//==============================================================
// 12) Brake release control
//==============================================================
// EN: A movement request keeps the magnetic brake released.
//     After movement stops, the brake remains released for a hold time.
conveyorLevelerMoveRequest :=
    systemRunEnable AND
    safetyCircuitOk AND
    conveyorLevelerDriveOk AND
    NOT conveyorLevelerFault AND
    (ABS(conveyorLevelerSignedSpeedRefMmps) >= machineConfig.conveyorLevelerRunMinSpeedMmps);


IF conveyorLevelerMoveRequest THEN

    conveyorLevelerBrakeReleaseRequest := TRUE;

    tonConveyorLevelerBrakeHoldDelay(IN := FALSE);

ELSE

    IF conveyorLevelerBrakeRelease THEN

        tonConveyorLevelerBrakeHoldDelay(
            IN := TRUE,
            PT := machineConfig.conveyorLevelerBrakeHoldTime
        );

        conveyorLevelerBrakeReleaseRequest :=
            NOT tonConveyorLevelerBrakeHoldDelay.Q;

    ELSE

        tonConveyorLevelerBrakeHoldDelay(IN := FALSE);
        conveyorLevelerBrakeReleaseRequest := FALSE;

    END_IF

END_IF;


conveyorLevelerBrakeRelease :=
    systemRunEnable AND
    safetyCircuitOk AND
    conveyorLevelerDriveOk AND
    NOT conveyorLevelerFault AND
    conveyorLevelerBrakeReleaseRequest;


//==============================================================
// 13) Brake release delay before motor movement
//==============================================================
// EN: The motor can run only after brake release delay.
tonConveyorLevelerBrakeReleaseDelay(
    IN := conveyorLevelerMoveRequest AND conveyorLevelerBrakeRelease,
    PT := machineConfig.conveyorLevelerBrakeReleaseDelay
);


//==============================================================
// 14) Conveyor leveler direction and speed outputs
//==============================================================
// EN: Convert signed internal speed command into direction outputs
//     and positive speed reference.
IF conveyorLevelerMoveRequest AND
   conveyorLevelerBrakeRelease AND
   tonConveyorLevelerBrakeReleaseDelay.Q THEN

    conveyorLevelerSpeedRefMmps :=
        ABS(conveyorLevelerSignedSpeedRefMmps);

    conveyorLevelerRunUp :=
        conveyorLevelerSignedSpeedRefMmps > 0.0;

    conveyorLevelerRunDown :=
        conveyorLevelerSignedSpeedRefMmps < 0.0;

ELSE

    conveyorLevelerSpeedRefMmps := 0.0;

    conveyorLevelerRunUp := FALSE;
    conveyorLevelerRunDown := FALSE;

END_IF;
END_METHOD

//==============================================================
// SIMPLE STACKER — SPEED REFERENCE GENERATOR
// EN: Generates synchronized and sheet-stack separation speed references [m/min].
//==============================================================
METHOD _ConveyorSpeedControl
VAR
    rPackageComplete                  : BOOL;
    packageGapReady                   : BOOL;
    validCycleTimeS                   : REAL;

    sheetConveyorsSpeedUpReferenceMPM : REAL;

    sheetConveyor1BaseSpeedMPM        : REAL;
    sheetConveyor2BaseSpeedMPM        : REAL;
    sheetConveyor3BaseSpeedMPM        : REAL;
END_VAR


//==============================================================
// 1) Default event pulses
//==============================================================
sheetStackSeparationStarted         := FALSE;
sheetStackSeparationFinished        := FALSE;

sheetConveyor2SeparationStarted     := FALSE;
sheetConveyor2SeparationFinished    := FALSE;

sheetConveyor3SeparationStarted     := FALSE;
sheetConveyor3SeparationFinished    := FALSE;


//==============================================================
// 2) Edge detection
//==============================================================
rPackageComplete := packageCompleteCmd AND NOT packageCompleteCmdOld;
packageCompleteCmdOld := packageCompleteCmd;


//==============================================================
// 3) Enable and scan time
//==============================================================
speedControlEnabled :=
    sheetConveyor1Run AND
    sheetConveyor2Run AND
    sheetConveyor3Run AND
    safetyCircuitOk;

rampReset := NOT speedControlEnabled;


// EN: Read PLC scan time using OSCAT CYCLE_TIME.
instCycleTime(
    RST := resetCmd
);


// EN: Convert last cycle time from TIME/ms to seconds.
scanTimeMs := TIME_TO_REAL(instCycleTime.ct_last);

validCycleTimeS :=
    LIMIT(
        0.001,
        scanTimeMs / 1000.0,
        20.0
    );

scanTimeS := validCycleTimeS;



//==============================================================
// 4) Calculate normal stacker speed
//==============================================================
IF speedControlEnabled THEN

    normalStackerSpeedMPM :=
        LIMIT(
            machineConfig.minimumSpeedMPM,
            MAX(0.0, lineSpeedMPM) *
                MAX(0.0, machineConfig.stackerSpeedRatio),
            machineConfig.maximumSpeedMPM
        );

ELSE

    normalStackerSpeedMPM := 0.0;

END_IF;


//==============================================================
// 6) Calculate normal speed for each conveyor
//==============================================================
sheetConveyor1NormalSpeedMPM :=
    normalStackerSpeedMPM *
    MAX(0.0, machineConfig.sheetConveyor1SpeedTrim);

sheetConveyor2NormalSpeedMPM :=
    normalStackerSpeedMPM *
    MAX(0.0, machineConfig.sheetConveyor2SpeedTrim);

sheetConveyor3NormalSpeedMPM :=
    normalStackerSpeedMPM *
    MAX(0.0, machineConfig.sheetConveyor3SpeedTrim);


//==============================================================
// 6.1) Sheet conveyors speed-up reference
//==============================================================
// EN: Speed-up is added directly to conveyors 1/2/3 references.
//     It can work even when line speed is zero, as long as the
//     conveyor group is enabled.
IF speedControlEnabled AND sheetConveyorsSpeedUpCmd THEN

    sheetConveyorsSpeedUpReferenceMPM :=
        MAX(0.0, machineConfig.sheetConveyorsSpeedUpMPM);

ELSE

    sheetConveyorsSpeedUpReferenceMPM := 0.0;

END_IF;


//==============================================================
// 6.2) Base speed references including speed-up
//==============================================================
// EN: Base speed is the synchronized conveyor speed plus operator speed-up.
//     Separation tracking must use this base speed as reference.
sheetConveyor1BaseSpeedMPM :=
    sheetConveyor1NormalSpeedMPM + sheetConveyorsSpeedUpReferenceMPM;

sheetConveyor2BaseSpeedMPM :=
    sheetConveyor2NormalSpeedMPM + sheetConveyorsSpeedUpReferenceMPM;

sheetConveyor3BaseSpeedMPM :=
    sheetConveyor3NormalSpeedMPM + sheetConveyorsSpeedUpReferenceMPM;


//==============================================================
// 7) Calculate separation high speed
//==============================================================
// EN: Gap speed also receives the same speed-up reference.
//     This preserves the real gap differential while allowing operator boost.
sheetConveyor2GapSpeedMPM :=
    (sheetConveyor2NormalSpeedMPM * MAX(0.0, machineConfig.packageGapSpeedRatio)) +
    machineConfig.packageGapSpeedOffsetMPM +
    sheetConveyorsSpeedUpReferenceMPM;

sheetConveyor3GapSpeedMPM :=
    (sheetConveyor3NormalSpeedMPM * MAX(0.0, machineConfig.packageGapSpeedRatio)) +
    machineConfig.packageGapSpeedOffsetMPM +
    sheetConveyorsSpeedUpReferenceMPM;


//==============================================================
// 8) Calculate separation tracking target distances
//==============================================================
// EN: Separation tracking target is based on each conveyor length.
sheetConveyor2TargetDistanceM :=
    MAX(0.0, machineConfig.sheetConveyor2LengthM);

sheetConveyor3TargetDistanceM :=
    MAX(0.0, machineConfig.sheetConveyor3LengthM);


//==============================================================
// 9) Check separation ready conditions
//==============================================================
// EN: Compare gap speed against base speed, not normal speed.
//     Otherwise operator speed-up would be incorrectly counted as gap opening.
packageGapReady :=
    speedControlEnabled AND
    (sheetConveyor2TargetDistanceM > 0.0) AND
    (sheetConveyor3TargetDistanceM > 0.0) AND
    ((sheetConveyor2GapSpeedMPM - sheetConveyor2BaseSpeedMPM) >= machineConfig.minimumOpeningSpeedMPM) AND
    ((sheetConveyor3GapSpeedMPM - sheetConveyor3BaseSpeedMPM) >= machineConfig.minimumOpeningSpeedMPM);

sheetStackSeparationReady := packageGapReady;


//==============================================================
// 10) Sheet stack separation state machine
//==============================================================
IF NOT speedControlEnabled THEN

    sheetStackSeparationState      := 'DISABLED';
    sheetStackSeparationStateCode  := -1;

    packageSeparationState         := 0;

    sheetStackSeparationActive     := FALSE;
    sheetStackBrakeActive          := FALSE;
    brakeValve                     := FALSE;

    sheetConveyor2SeparationActive := FALSE;
    sheetConveyor3SeparationActive := FALSE;

    sheetConveyor2HighSpeedActive  := FALSE;
    sheetConveyor3HighSpeedActive  := FALSE;

    sheetConveyor2OpeningDistanceM := 0.0;
    sheetConveyor3OpeningDistanceM := 0.0;

    sheetConveyor1TargetSpeedMPM   := 0.0;
    sheetConveyor2TargetSpeedMPM   := 0.0;
    sheetConveyor3TargetSpeedMPM   := 0.0;


ELSE

    CASE packageSeparationState OF

        0: // NORMAL
            sheetStackSeparationState     := 'NORMAL';
            sheetStackSeparationStateCode := 0;

            sheetStackSeparationActive    := FALSE;
            sheetStackBrakeActive         := FALSE;
            brakeValve                    := FALSE;

            sheetConveyor2SeparationActive := FALSE;
            sheetConveyor3SeparationActive := FALSE;

            sheetConveyor2HighSpeedActive  := FALSE;
            sheetConveyor3HighSpeedActive  := FALSE;

            sheetConveyor2OpeningDistanceM := 0.0;
            sheetConveyor3OpeningDistanceM := 0.0;

            sheetConveyor1TargetSpeedMPM  := sheetConveyor1BaseSpeedMPM;
            sheetConveyor2TargetSpeedMPM  := sheetConveyor2BaseSpeedMPM;
            sheetConveyor3TargetSpeedMPM  := sheetConveyor3BaseSpeedMPM;

            IF rPackageComplete AND packageGapReady THEN
                packageSeparationState := 10;
            END_IF


        10: // START_SHEET_STACK_SEPARATION
            sheetStackSeparationState     := 'START_SEPARATION';
            sheetStackSeparationStateCode := 10;

            sheetStackSeparationActive    := TRUE;
            sheetStackSeparationStarted   := TRUE;

            sheetStackBrakeActive         := TRUE;
            brakeValve                    := TRUE;

            // EN: Conveyor 2 tracking starts immediately.
            sheetConveyor2SeparationStarted := TRUE;

            sheetConveyor2SeparationActive  := TRUE;
            sheetConveyor3SeparationActive  := FALSE;

            // EN: Conveyor 2 and 3 accelerate together from the beginning.
            sheetConveyor2HighSpeedActive   := TRUE;
            sheetConveyor3HighSpeedActive   := TRUE;

            sheetConveyor2OpeningDistanceM  := 0.0;
            sheetConveyor3OpeningDistanceM  := 0.0;

            sheetConveyor1TargetSpeedMPM    := sheetConveyor1BaseSpeedMPM;
            sheetConveyor2TargetSpeedMPM    := sheetConveyor2GapSpeedMPM;
            sheetConveyor3TargetSpeedMPM    := sheetConveyor3GapSpeedMPM;

            packageSeparationState := 20;


        20: // SHEET_CONVEYOR_2_SEPARATION_TRACKING
            sheetStackSeparationState     := 'CONV2_TRACKING';
            sheetStackSeparationStateCode := 20;

            sheetStackSeparationActive    := TRUE;

            sheetStackBrakeActive         := TRUE;
            brakeValve                    := TRUE;

            sheetConveyor2SeparationActive := TRUE;
            sheetConveyor3SeparationActive := FALSE;

            sheetConveyor2HighSpeedActive  := TRUE;
            sheetConveyor3HighSpeedActive  := TRUE;

            sheetConveyor1TargetSpeedMPM  := sheetConveyor1BaseSpeedMPM;
            sheetConveyor2TargetSpeedMPM  := sheetConveyor2GapSpeedMPM;
            sheetConveyor3TargetSpeedMPM  := sheetConveyor3GapSpeedMPM;

            IF sheetConveyor2OpeningDistanceM >= sheetConveyor2TargetDistanceM THEN

                // EN: Conveyor 2 tracking finished. Conveyor 2 returns to base speed.
                sheetConveyor2SeparationFinished := TRUE;

                sheetConveyor2SeparationActive   := FALSE;
                sheetConveyor2HighSpeedActive    := FALSE;

                sheetStackBrakeActive            := FALSE;
                brakeValve                       := FALSE;

                sheetConveyor2TargetSpeedMPM     := sheetConveyor2BaseSpeedMPM;

                // EN: Conveyor 3 tracking starts after conveyor 2 returns to sync.
                sheetConveyor3SeparationStarted := TRUE;
                sheetConveyor3OpeningDistanceM  := 0.0;

                packageSeparationState := 30;

            END_IF


        30: // SHEET_CONVEYOR_3_SEPARATION_TRACKING
            sheetStackSeparationState     := 'CONV3_TRACKING';
            sheetStackSeparationStateCode := 30;

            sheetStackSeparationActive    := TRUE;

            sheetStackBrakeActive         := FALSE;
            brakeValve                    := FALSE;

            sheetConveyor2SeparationActive := FALSE;
            sheetConveyor3SeparationActive := TRUE;

            sheetConveyor2HighSpeedActive  := FALSE;
            sheetConveyor3HighSpeedActive  := TRUE;

            sheetConveyor1TargetSpeedMPM  := sheetConveyor1BaseSpeedMPM;
            sheetConveyor2TargetSpeedMPM  := sheetConveyor2BaseSpeedMPM;
            sheetConveyor3TargetSpeedMPM  := sheetConveyor3GapSpeedMPM;

            IF sheetConveyor3OpeningDistanceM >= sheetConveyor3TargetDistanceM THEN

                // EN: Conveyor 3 returns to base synchronized speed.
                sheetConveyor3TargetSpeedMPM := sheetConveyor3BaseSpeedMPM;

                packageSeparationState := 40;

            END_IF


        40: // FINISH_SHEET_STACK_SEPARATION
            sheetStackSeparationState     := 'FINISH_SEPARATION';
            sheetStackSeparationStateCode := 40;

            sheetStackSeparationActive    := FALSE;
            sheetStackSeparationFinished  := TRUE;

            sheetStackBrakeActive         := FALSE;
            brakeValve                    := FALSE;

            sheetConveyor2SeparationActive  := FALSE;
            sheetConveyor3SeparationActive  := FALSE;

            sheetConveyor2HighSpeedActive   := FALSE;
            sheetConveyor3HighSpeedActive   := FALSE;

            sheetConveyor3SeparationFinished := TRUE;

            sheetConveyor1TargetSpeedMPM  := sheetConveyor1BaseSpeedMPM;
            sheetConveyor2TargetSpeedMPM  := sheetConveyor2BaseSpeedMPM;
            sheetConveyor3TargetSpeedMPM  := sheetConveyor3BaseSpeedMPM;

            packageSeparationState := 0;


    ELSE

        packageSeparationState := 0;

    END_CASE;

END_IF;


//==============================================================
// 11) Limit speed targets
//==============================================================
sheetConveyor1TargetSpeedMPM := LIMIT(
    machineConfig.minimumSpeedMPM,
    sheetConveyor1TargetSpeedMPM,
    machineConfig.maximumSpeedMPM
);

sheetConveyor2TargetSpeedMPM := LIMIT(
    machineConfig.minimumSpeedMPM,
    sheetConveyor2TargetSpeedMPM,
    machineConfig.maximumSpeedMPM
);

sheetConveyor3TargetSpeedMPM := LIMIT(
    machineConfig.minimumSpeedMPM,
    sheetConveyor3TargetSpeedMPM,
    machineConfig.maximumSpeedMPM
);


//==============================================================
// 12) Ramp sheet conveyor 1 speed reference
//==============================================================
instRampSheetConveyor1(
    X          := sheetConveyor1TargetSpeedMPM,
    A_UP       := MAX(0.0, machineConfig.rampAccelerationUpMPMps2),
    A_DN       := -MAX(0.0, machineConfig.rampAccelerationDownMPMps2),
    VU_MAX     := MAX(0.0, machineConfig.rampVelocityUpMaxMPMps),
    VD_MAX     := -MAX(0.0, machineConfig.rampVelocityDownMaxMPMps),
    LIMIT_HIGH := machineConfig.maximumSpeedMPM,
    LIMIT_LOW  := machineConfig.minimumSpeedMPM,
    RST        := rampReset,
    Y          => sheetConveyor1SpeedRefMPM
);


//==============================================================
// 13) Ramp sheet conveyor 2 speed reference
//==============================================================
instRampSheetConveyor2(
    X          := sheetConveyor2TargetSpeedMPM,
    A_UP       := MAX(0.0, machineConfig.rampAccelerationUpMPMps2),
    A_DN       := -MAX(0.0, machineConfig.rampAccelerationDownMPMps2),
    VU_MAX     := MAX(0.0, machineConfig.rampVelocityUpMaxMPMps),
    VD_MAX     := -MAX(0.0, machineConfig.rampVelocityDownMaxMPMps),
    LIMIT_HIGH := machineConfig.maximumSpeedMPM,
    LIMIT_LOW  := machineConfig.minimumSpeedMPM,
    RST        := rampReset,
    Y          => sheetConveyor2SpeedRefMPM
);


//==============================================================
// 14) Ramp sheet conveyor 3 speed reference
//==============================================================
instRampSheetConveyor3(
    X          := sheetConveyor3TargetSpeedMPM,
    A_UP       := MAX(0.0, machineConfig.rampAccelerationUpMPMps2),
    A_DN       := -MAX(0.0, machineConfig.rampAccelerationDownMPMps2),
    VU_MAX     := MAX(0.0, machineConfig.rampVelocityUpMaxMPMps),
    VD_MAX     := -MAX(0.0, machineConfig.rampVelocityDownMaxMPMps),
    LIMIT_HIGH := machineConfig.maximumSpeedMPM,
    LIMIT_LOW  := machineConfig.minimumSpeedMPM,
    RST        := rampReset,
    Y          => sheetConveyor3SpeedRefMPM
);


//==============================================================
// 16) Calculate real separation tracking speed using ramped references
//==============================================================
// EN: Only the real speed differential above the base speed moves the
//     separation point through the conveyors.
//     Operator speed-up is already included in base speed, so it is not
//     counted as gap opening.
sheetConveyor2OpeningSpeedMPM :=
    MAX(0.0, sheetConveyor2SpeedRefMPM - sheetConveyor2BaseSpeedMPM);

sheetConveyor3OpeningSpeedMPM :=
    MAX(0.0, sheetConveyor3SpeedRefMPM - sheetConveyor3BaseSpeedMPM);


//==============================================================
// 17) Integrate real separation tracking distance
//==============================================================
IF speedControlEnabled THEN

    IF packageSeparationState = 20 THEN

        IF sheetConveyor2OpeningSpeedMPM >= machineConfig.minimumOpeningSpeedMPM THEN

            sheetConveyor2OpeningDistanceM :=
                sheetConveyor2OpeningDistanceM +
                (sheetConveyor2OpeningSpeedMPM / 60.0) * scanTimeS;

        END_IF

    ELSIF packageSeparationState = 30 THEN

        IF sheetConveyor3OpeningSpeedMPM >= machineConfig.minimumOpeningSpeedMPM THEN

            sheetConveyor3OpeningDistanceM :=
                sheetConveyor3OpeningDistanceM +
                (sheetConveyor3OpeningSpeedMPM / 60.0) * scanTimeS;

        END_IF

    END_IF

END_IF;


//==============================================================
// 18) Publish tracking distances to outputs
//==============================================================
sheetConveyor2TrackingDistanceM := sheetConveyor2OpeningDistanceM;
sheetConveyor3TrackingDistanceM := sheetConveyor3OpeningDistanceM;
END_METHOD

//==============================================================
// SIMPLE STACKER — HMI STATUS
// EN: Maps internal status, outputs, positions and diagnostics
//     to the HMI status structure.
//==============================================================
METHOD _HmiStatus



//==============================================================
// 1) System general status
//==============================================================
hmiStatus.systemRunEnable :=
    systemRunEnable;

hmiStatus.safetyCircuitOk :=
    safetyCircuitOk;

hmiStatus.faultActive :=
    faultActive OR
    backstopFault OR
    conveyorLevelerFault OR
    sheetStackDischargeFault OR
    sheetStackDischargeConveyorFault;

hmiStatus.deviceState :=
    deviceState;


//==============================================================
// 2) Sheet conveyor group status
//==============================================================
hmiStatus.synchronizedConveyorsRunning :=
    synchronizedConveyorsRunning;

hmiStatus.sheetConveyor1Run :=
    sheetConveyor1Run;

hmiStatus.sheetConveyor2Run :=
    sheetConveyor2Run;

hmiStatus.sheetConveyor3Run :=
    sheetConveyor3Run;

hmiStatus.sheetConveyor1SpeedRefMPM :=
    sheetConveyor1SpeedRefMPM;

hmiStatus.sheetConveyor2SpeedRefMPM :=
    sheetConveyor2SpeedRefMPM;

hmiStatus.sheetConveyor3SpeedRefMPM :=
    sheetConveyor3SpeedRefMPM;

hmiStatus.syncConveyorsState :=
    syncConveyorsState;


//==============================================================
// 3) Sheet stack separation status
//==============================================================
hmiStatus.sheetStackSeparationReady :=
    sheetStackSeparationReady;

hmiStatus.sheetStackSeparationActive :=
    sheetStackSeparationActive;

hmiStatus.sheetStackBrakeActive :=
    sheetStackBrakeActive;


//==============================================================
// 4) Sheet stack discharge sequence status
//==============================================================
hmiStatus.sheetStackDischargeState :=
    sheetStackDischargeState;

hmiStatus.sheetStackDischargeStateCode :=
    sheetStackDischargeStateCode;

hmiStatus.sheetStackDischargePending :=
    sheetStackDischargePending;

hmiStatus.sheetStackDischargeActive :=
    sheetStackDischargeActive;

hmiStatus.sheetStackDischargeStarted :=
    sheetStackDischargeStarted;

hmiStatus.sheetStackDischargeFinished :=
    sheetStackDischargeFinished;

hmiStatus.sheetStackDischargeFault :=
    sheetStackDischargeFault;

hmiStatus.sheetStackDischargeFaultCode :=
    sheetStackDischargeFaultCode;

hmiStatus.sheetStackDischargeLastCycleOk :=
    sheetStackDischargeLastCycleOk;

hmiStatus.sheetStackDischargeLastResultCode :=
    sheetStackDischargeLastResultCode;

hmiStatus.sheetStackDischargeLastFaultStepCode :=
    sheetStackDischargeLastFaultStepCode;

hmiStatus.sheetStackDischargeLastFaultCode :=
    sheetStackDischargeLastFaultCode;


//==============================================================
// 5) Sheet stack discharge conveyor status
//==============================================================
hmiStatus.sheetStackDischargeConveyorState :=
    sheetStackDischargeConveyorState;

hmiStatus.sheetStackDischargeConveyorRun :=
    sheetStackDischargeConveyorRun;

hmiStatus.sheetStackDischargeConveyorSpeedRefMPM :=
    sheetStackDischargeConveyorSpeedRefMPM;

hmiStatus.sheetStackDischargeConveyorFault :=
    sheetStackDischargeConveyorFault;

hmiStatus.sheetStackDischargeConveyorFaultCode :=
    sheetStackDischargeConveyorFaultCode;


//==============================================================
// 6) Backstop status
//==============================================================
hmiStatus.backstopState :=
    backstopState;

hmiStatus.backstopHomed :=
    backstopHomed;

hmiStatus.backstopHomeRunning :=
    backstopHomeRunning;

hmiStatus.backstopInPosition :=
    backstopInPosition;

hmiStatus.backstopPositionMm :=
    backstopPositionMm;

hmiStatus.backstopTargetPositionMm :=
    backstopTargetPositionMm;

hmiStatus.backstopPositionErrorMm :=
    backstopPositionErrorMm;

hmiStatus.backstopRunFw :=
    backstopRunFw;

hmiStatus.backstopRunRev :=
    backstopRunRev;

hmiStatus.backstopSpeedRefMmps :=
    backstopSpeedRefMmps;

hmiStatus.backstopPlateUpSolenoid :=
    backstopPlateUpSolenoid;

hmiStatus.backstopSetEncoderPosition :=
    backstopSetEncoderPosition;

hmiStatus.backstopSetEncoderPositionMm :=
    backstopSetEncoderPositionMm;

hmiStatus.backstopManualInterventionActive :=
    backstopManualInterventionActive;

hmiStatus.backstopManualInterventionPositionMm :=
    backstopManualInterventionPositionMm;

hmiStatus.backstopFault :=
    backstopFault;

hmiStatus.backstopFaultCode :=
    backstopFaultCode;


//==============================================================
// 7) Conveyor leveler status
//==============================================================
hmiStatus.conveyorLevelerState :=
    conveyorLevelerState;

hmiStatus.conveyorLevelerHomed :=
    conveyorLevelerHomed;

hmiStatus.conveyorLevelerInPosition :=
    conveyorLevelerInPosition;

hmiStatus.conveyorLevelerPositionMm :=
    conveyorLevelerPositionMm;

hmiStatus.conveyorLevelerTargetPositionMm :=
    conveyorLevelerTargetPositionMm;

hmiStatus.conveyorLevelerPositionErrorMm :=
    conveyorLevelerPositionErrorMm;

hmiStatus.conveyorLevelerRunUp :=
    conveyorLevelerRunUp;

hmiStatus.conveyorLevelerRunDown :=
    conveyorLevelerRunDown;

hmiStatus.conveyorLevelerBrakeRelease :=
    conveyorLevelerBrakeRelease;

hmiStatus.conveyorLevelerSpeedRefMmps :=
    conveyorLevelerSpeedRefMmps;

hmiStatus.conveyorLevelerSetEncoderPosition :=
    conveyorLevelerSetEncoderPosition;

hmiStatus.conveyorLevelerSetEncoderPositionMm :=
    conveyorLevelerSetEncoderPositionMm;

hmiStatus.conveyorLevelerFault :=
    conveyorLevelerFault;

hmiStatus.conveyorLevelerFaultCode :=
    conveyorLevelerFaultCode;


//==============================================================
// 8) Process values
//==============================================================
hmiStatus.lineSpeedMPM :=
    lineSpeedMPM;

hmiStatus.sheetLengthMm :=
    sheetLengthMm;

hmiStatus.stackHeightMm :=
    stackHeightMm;


//==============================================================
// 9) Input / drive status mirror
//==============================================================
hmiStatus.sheetConveyor1DriveOk :=
    sheetConveyor1DriveOk;

hmiStatus.sheetConveyor2DriveOk :=
    sheetConveyor2DriveOk;

hmiStatus.sheetConveyor3DriveOk :=
    sheetConveyor3DriveOk;

hmiStatus.backstopDriveOk :=
    backstopDriveOk;

hmiStatus.conveyorLevelerDriveOk :=
    conveyorLevelerDriveOk;

hmiStatus.sheetStackDischargeConveyorDriveOk :=
    sheetStackDischargeConveyorDriveOk;
END_METHOD

METHOD _MachineAuxiliary
VAR_INPUT
END_VAR
(*



stopMachinePulse :=
    NOT safetyCircuitOk OR
    NOT sheetConveyor1DriveOk OR
    NOT sheetConveyor2DriveOk OR
    NOT sheetConveyor3DriveOk;
	NOT backstopDriveOk
	NOT conveyorLevelerDriveOk
*)
noCrushRollersUpDownValve := noCrushRollersDownCmd;

stackerRunning := systemRunEnable;


reset := resetCmd;
END_METHOD

//==============================================================
// SIMPLE STACKER — SHEET CONVEYOR GROUP CONTROL
// EN: Controls the synchronized sheet conveyor group.
//     Start/stop command latch is handled by _SystemControl().
//==============================================================
METHOD _SheetConveyorGroupControl

//==============================================================
// 1) Conditions
//==============================================================
// EN: Only synchronized sheet conveyor drives are considered here.
// PT: Apenas os inversores das esteiras sincronizadas são considerados aqui.
allSynchronizedDrivesOk :=
    sheetConveyor1DriveOk AND
    sheetConveyor2DriveOk AND
    sheetConveyor3DriveOk;


// EN: Synchronized conveyor group fault.
// PT: Falha do grupo de esteiras sincronizadas.
anyFault :=
    NOT safetyCircuitOk OR
    NOT allSynchronizedDrivesOk;

faultActive := anyFault;


//==============================================================
// 2) State machine
//==============================================================
CASE syncConveyorsState OF

    0: // IDLE
        deviceState := 'IDLE';

        sheetConveyor1Run := FALSE;
        sheetConveyor2Run := FALSE;
        sheetConveyor3Run := FALSE;

        synchronizedConveyorsRunning := FALSE;

        // EN: The group starts only when the master system is enabled
        //     and no conveyor group fault is active.
        IF systemRunEnable AND NOT anyFault THEN

            syncConveyorsState := 1;

        ELSIF systemRunEnable AND anyFault THEN

            syncConveyorsState := 10;

        END_IF


    1: // RUN
        deviceState := 'RUN';

        // EN: Outputs are also directly conditioned by systemRunEnable
        //     to avoid one-scan movement after a stop command.
        sheetConveyor1Run :=
            systemRunEnable AND
            safetyCircuitOk AND
            sheetConveyor1DriveOk;

        sheetConveyor2Run :=
            systemRunEnable AND
            safetyCircuitOk AND
            sheetConveyor2DriveOk;

        sheetConveyor3Run :=
            systemRunEnable AND
            safetyCircuitOk AND
            sheetConveyor3DriveOk;

        synchronizedConveyorsRunning :=
            sheetConveyor1Run AND
            sheetConveyor2Run AND
            sheetConveyor3Run;

        IF anyFault THEN

            syncConveyorsState := 10;

        ELSIF NOT systemRunEnable THEN

            syncConveyorsState := 0;

        END_IF


    10: // FAULT
        deviceState := 'FAULT';

        sheetConveyor1Run := FALSE;
        sheetConveyor2Run := FALSE;
        sheetConveyor3Run := FALSE;

        synchronizedConveyorsRunning := FALSE;

        // EN: Fault state is released only by reset and with all faults cleared.
        //     If systemRunEnable is still TRUE after reset, the group can start
        //     again from IDLE on the next scan.
        IF resetCmd AND NOT anyFault THEN

            syncConveyorsState := 0;

        END_IF


ELSE

    syncConveyorsState := 0;

END_CASE;
END_METHOD

//==============================================================
// SIMPLE STACKER — SHEET STACK DISCHARGE CONTROL
// EN: Controls the sheet stack discharge sequence after the sheet
//     conveyor separation cycle is completed.
//
// State code
// 0  = IDLE
// 5  = WAIT_SEPARATION
// 10 = START_DISCHARGE_POSITIONING
// 20 = WAIT_BACKSTOP_POSITION
// 30 = RUN_DISCHARGE_CONVEYOR
// 40 = START_RETURN_POSITIONING
// 50 = WAIT_BACKSTOP_RETURN
// 60 = FINISH
// 90 = ABORT_TRANSIENT
//
// Last result code
// 0 = No cycle executed yet
// 1 = Last cycle completed successfully
// 2 = Last cycle completed with manual backstop skip
// 3 = Last cycle completed/aborted by timeout
// 4 = Last cycle aborted by fault
//
// Fault code
// 0  = No fault
// 1  = Safety circuit not OK
// 2  = Sheet conveyor drive not OK
// 3  = Discharge conveyor drive/control fault
// 4  = Backstop drive/control fault
// 5  = Conveyor leveler drive/control fault
// 6  = Stacker stopped during cycle
// 10 = Wait separation timeout
// 20 = Backstop positioning timeout
// 30 = Discharge conveyor did not start timeout
// 50 = Backstop return timeout
//==============================================================
METHOD _SheetStackDischargeControl
VAR
    abortCycle : BOOL;
END_VAR


//==============================================================
// 1) Default event pulses
//==============================================================
sheetStackDischargeStarted  := FALSE;
sheetStackDischargeFinished := FALSE;


//==============================================================
// 2) Default internal requests / overrides
//==============================================================
// EN: The sequence does not write the physical discharge conveyor outputs.
//     It only generates an internal request to the conveyor control method.
sheetStackDischargeConveyorRunRequest := FALSE;

backstopTargetOverrideActive := FALSE;
backstopTargetOverridePositionMm := 0.0;

conveyorLevelerTargetOverrideActive := FALSE;
conveyorLevelerTargetOverridePositionMm := 0.0;


//==============================================================
// 3) Edge detection
//==============================================================
// EN: Separate edge detector to avoid interfering with conveyor speed control.
rPackageCompleteDischarge :=
    packageCompleteCmd AND NOT packageCompleteCmdOldDischarge;

packageCompleteCmdOldDischarge := packageCompleteCmd;


//==============================================================
// 4) Fault condition
//==============================================================
// EN: Conveyor leveler feedback is not used for sequence progress,
//     but its drive/control fault still aborts the cycle.
sheetStackDischargeFaultCondition :=
    NOT safetyCircuitOk OR
    NOT sheetConveyor1DriveOk OR
    NOT sheetConveyor2DriveOk OR
    NOT sheetConveyor3DriveOk OR
    NOT sheetStackDischargeConveyorDriveOk OR
    sheetStackDischargeConveyorFault OR
    NOT backstopDriveOk OR
    backstopFault OR
    NOT conveyorLevelerDriveOk OR
    conveyorLevelerFault;


//==============================================================
// 5) Fault code priority
//==============================================================
IF NOT safetyCircuitOk THEN

    sheetStackDischargeFaultCode := 1;

ELSIF NOT sheetConveyor1DriveOk OR
      NOT sheetConveyor2DriveOk OR
      NOT sheetConveyor3DriveOk THEN

    sheetStackDischargeFaultCode := 2;

ELSIF NOT sheetStackDischargeConveyorDriveOk OR
      sheetStackDischargeConveyorFault THEN

    sheetStackDischargeFaultCode := 3;

ELSIF NOT backstopDriveOk OR
      backstopFault THEN

    sheetStackDischargeFaultCode := 4;

ELSIF NOT conveyorLevelerDriveOk OR
      conveyorLevelerFault THEN

    sheetStackDischargeFaultCode := 5;

ELSIF NOT synchronizedConveyorsRunning THEN

    sheetStackDischargeFaultCode := 6;

END_IF;


//==============================================================
// 6) Optional reset of current sequence fault display
//==============================================================
// EN: Reset clears the current sequence fault flag,
//     but does not erase last cycle diagnostic codes.
IF resetCmd AND (sheetStackDischargeControlState = 0) THEN

    sheetStackDischargeFault := FALSE;
    sheetStackDischargeFaultCode := 0;

END_IF;


//==============================================================
// 7) Arm discharge sequence from packageCompleteCmd
//==============================================================
// EN: packageCompleteCmd is ignored if stacker is not running or if
//     any relevant drive/safety fault is active.
IF rPackageCompleteDischarge AND
   synchronizedConveyorsRunning AND
   NOT sheetStackDischargeFaultCondition AND
   NOT sheetStackDischargeActive AND
   NOT sheetStackDischargePending THEN

    sheetStackDischargePending := TRUE;

    // EN: Clear current-cycle flags when a new cycle is accepted.
    sheetStackDischargeFault := FALSE;
    sheetStackDischargeFaultCode := 0;

    sheetStackDischargeCycleHasManualSkip := FALSE;
    sheetStackDischargeCycleHasTimeout := FALSE;

END_IF;


//==============================================================
// 8) Immediate abort condition
//==============================================================
// EN: Any relevant fault during an active/pending cycle aborts the
//     sequence and automatically returns to IDLE.
//     Loss of synchronized conveyor running also aborts the cycle.
abortCycle :=
    (
        sheetStackDischargeActive OR
        sheetStackDischargePending OR
        (sheetStackDischargeControlState <> 0)
    )
    AND
    (
        sheetStackDischargeFaultCondition OR
        NOT synchronizedConveyorsRunning
    );


IF abortCycle THEN

    sheetStackDischargeConveyorRunRequest := FALSE;

    backstopTargetOverrideActive := FALSE;
    conveyorLevelerTargetOverrideActive := FALSE;

    sheetStackDischargePending := FALSE;
    sheetStackDischargeActive := FALSE;

    tonSheetStackDischarge(IN := FALSE);
    tonSheetStackDischargeStepTimeout(IN := FALSE);

    sheetStackDischargeFault := TRUE;

    sheetStackDischargeLastCycleOk := FALSE;
    sheetStackDischargeLastResultCode := 4;
    sheetStackDischargeLastFaultStepCode := sheetStackDischargeControlState;
    sheetStackDischargeLastFaultCode := sheetStackDischargeFaultCode;

    sheetStackDischargeState := 'ABORTED';
    sheetStackDischargeStateCode := 90;

    // EN: Do not clear backstopManualInterventionActive here.
    //     If the cycle aborted before return, keeping the memory is safer
    //     for the next cycle.

    // EN: No latched FAULT state. Return to IDLE automatically.
    sheetStackDischargeControlState := 0;


ELSE

    //==============================================================
    // 9) Sheet stack discharge state machine
    //==============================================================
    CASE sheetStackDischargeControlState OF

        0: // IDLE
            sheetStackDischargeState := 'IDLE';
            sheetStackDischargeStateCode := 0;

            sheetStackDischargeActive := FALSE;

            sheetStackDischargeConveyorRunRequest := FALSE;

            backstopTargetOverrideActive := FALSE;
            conveyorLevelerTargetOverrideActive := FALSE;

            tonSheetStackDischarge(IN := FALSE);
            tonSheetStackDischargeStepTimeout(IN := FALSE);

            IF sheetStackDischargePending THEN

                tonSheetStackDischarge(IN := FALSE);
                tonSheetStackDischargeStepTimeout(IN := FALSE);

                sheetStackDischargeControlState := 5;

            END_IF


        5: // WAIT_SEPARATION
            sheetStackDischargeState := 'WAIT_SEPARATION';
            sheetStackDischargeStateCode := 5;

            sheetStackDischargeActive := FALSE;

            sheetStackDischargeConveyorRunRequest := FALSE;

            backstopTargetOverrideActive := FALSE;
            conveyorLevelerTargetOverrideActive := FALSE;

            tonSheetStackDischarge(IN := FALSE);

            // EN: Wait for conveyor speed control to finish sheet stack separation.
            tonSheetStackDischargeStepTimeout(
                IN := TRUE,
                PT := machineConfig.sheetStackDischargeWaitSeparationTimeout
            );

            IF sheetStackSeparationFinished THEN

                tonSheetStackDischargeStepTimeout(IN := FALSE);

                sheetStackDischargeControlState := 10;


            ELSIF tonSheetStackDischargeStepTimeout.Q THEN

                // EN: Separation did not finish. Do not discharge.
                tonSheetStackDischargeStepTimeout(IN := FALSE);

                sheetStackDischargePending := FALSE;
                sheetStackDischargeActive := FALSE;

                sheetStackDischargeFault := TRUE;
                sheetStackDischargeFaultCode := 10;

                sheetStackDischargeLastCycleOk := FALSE;
                sheetStackDischargeLastResultCode := 3;
                sheetStackDischargeLastFaultStepCode := 5;
                sheetStackDischargeLastFaultCode := 10;

                sheetStackDischargeControlState := 0;

            END_IF


        10: // START_DISCHARGE_POSITIONING
            sheetStackDischargeState := 'START_POSITIONING';
            sheetStackDischargeStateCode := 10;

            sheetStackDischargePending := FALSE;
            sheetStackDischargeActive := TRUE;
            sheetStackDischargeStarted := TRUE;

            tonSheetStackDischarge(IN := FALSE);
            tonSheetStackDischargeStepTimeout(IN := FALSE);

            //======================================================
            // EN: Latch programmed backstop target for this cycle.
            //     This is the normal position based on sheet length.
            //======================================================
            backstopProgrammedDischargeTargetMm :=
                LIMIT(
                    machineConfig.backstopMinPositionMm,
                    MAX(0.0, sheetLengthMm) +
                        machineConfig.backstopSheetLengthOffsetMm,
                    machineConfig.backstopMaxPositionMm
                );

            //======================================================
            // EN: Define safe opening base position.
            //
            // If the operator manually moved the backstop before the
            // automatic cycle, use the greater value between:
            // - programmed position
            // - last manual intervention position
            //
            // This prevents the automatic opening override from closing
            // the backstop onto the material.
            //
            // If there was no manual intervention, use only the programmed
            // position as the base.
            //======================================================
            IF backstopManualInterventionActive THEN

                backstopDischargeOpenBasePositionMm :=
                    MAX(
                        backstopProgrammedDischargeTargetMm,
                        backstopManualInterventionPositionMm
                    );

            ELSE

                backstopDischargeOpenBasePositionMm :=
                    backstopProgrammedDischargeTargetMm;

            END_IF;

            //======================================================
            // EN: Latch safe discharge open target.
            //     Offset is applied after selecting the safe base.
            //======================================================
            backstopDischargeOpenTargetMm :=
                LIMIT(
                    machineConfig.backstopMinPositionMm,
                    backstopDischargeOpenBasePositionMm +
                        machineConfig.backstopDischargeOpenOffsetMm,
                    machineConfig.backstopMaxPositionMm
                );

            // EN: Request safe backstop opening.
            //     Backstop control accepts it only in auto.
            backstopTargetOverrideActive := TRUE;
            backstopTargetOverridePositionMm := backstopDischargeOpenTargetMm;

            // EN: Request conveyor leveler to move up.
            //     The sequence does not wait for leveler feedback.
            conveyorLevelerTargetOverrideActive := TRUE;
            conveyorLevelerTargetOverridePositionMm :=
                machineConfig.conveyorLevelerMaxPositionMm;

            sheetStackDischargeControlState := 20;


        20: // WAIT_BACKSTOP_POSITION
            sheetStackDischargeState := 'WAIT_BACKSTOP_POSITION';
            sheetStackDischargeStateCode := 20;

            sheetStackDischargeActive := TRUE;

            // EN: Keep safe latched backstop discharge target active.
            backstopTargetOverrideActive := TRUE;
            backstopTargetOverridePositionMm := backstopDischargeOpenTargetMm;

            // EN: Keep conveyor leveler up target active.
            //     Feedback is intentionally ignored for sequence progress.
            conveyorLevelerTargetOverrideActive := TRUE;
            conveyorLevelerTargetOverridePositionMm :=
                machineConfig.conveyorLevelerMaxPositionMm;

            // EN: If backstop is not in auto, do not wait for it.
            IF NOT backstopAutoCmd THEN

                sheetStackDischargeCycleHasManualSkip := TRUE;

                tonSheetStackDischargeStepTimeout(IN := FALSE);

                sheetStackDischargeControlState := 30;


            ELSIF backstopInPosition THEN

                tonSheetStackDischargeStepTimeout(IN := FALSE);

                sheetStackDischargeControlState := 30;


            ELSE

                tonSheetStackDischargeStepTimeout(
                    IN := TRUE,
                    PT := machineConfig.sheetStackDischargePositioningTimeout
                );

                IF tonSheetStackDischargeStepTimeout.Q THEN

                    // EN: Do not stay trapped waiting for backstop.
                    //     Continue the cycle, but record timeout diagnostic.
                    tonSheetStackDischargeStepTimeout(IN := FALSE);

                    sheetStackDischargeCycleHasTimeout := TRUE;

                    sheetStackDischargeFault := TRUE;
                    sheetStackDischargeFaultCode := 20;

                    sheetStackDischargeLastCycleOk := FALSE;
                    sheetStackDischargeLastResultCode := 3;
                    sheetStackDischargeLastFaultStepCode := 20;
                    sheetStackDischargeLastFaultCode := 20;

                    sheetStackDischargeControlState := 30;

                END_IF

            END_IF


        30: // RUN_DISCHARGE_CONVEYOR
            sheetStackDischargeState := 'DISCHARGING';
            sheetStackDischargeStateCode := 30;

            sheetStackDischargeActive := TRUE;

            // EN: Keep safe latched backstop discharge target active
            //     while discharging.
            backstopTargetOverrideActive := TRUE;
            backstopTargetOverridePositionMm := backstopDischargeOpenTargetMm;

            // EN: Keep conveyor leveler up while discharging.
            conveyorLevelerTargetOverrideActive := TRUE;
            conveyorLevelerTargetOverridePositionMm :=
                machineConfig.conveyorLevelerMaxPositionMm;

            // EN: Request discharge conveyor run.
            //     Physical output is controlled by _SheetStackDischargeConveyorControl.
            sheetStackDischargeConveyorRunRequest := TRUE;

            // EN: If conveyor is not actually running, use start timeout.
            IF NOT sheetStackDischargeConveyorRun THEN

                tonSheetStackDischarge(IN := FALSE);

                tonSheetStackDischargeStepTimeout(
                    IN := TRUE,
                    PT := machineConfig.sheetStackDischargeConveyorStartTimeout
                );

                IF tonSheetStackDischargeStepTimeout.Q THEN

                    // EN: Conveyor did not start. Do not stay trapped.
                    tonSheetStackDischargeStepTimeout(IN := FALSE);

                    sheetStackDischargeConveyorRunRequest := FALSE;

                    sheetStackDischargeCycleHasTimeout := TRUE;

                    sheetStackDischargeFault := TRUE;
                    sheetStackDischargeFaultCode := 30;

                    sheetStackDischargeLastCycleOk := FALSE;
                    sheetStackDischargeLastResultCode := 3;
                    sheetStackDischargeLastFaultStepCode := 30;
                    sheetStackDischargeLastFaultCode := 30;

                    sheetStackDischargeControlState := 40;

                END_IF


            ELSE

                // EN: Conveyor is running. Count real discharge time.
                tonSheetStackDischargeStepTimeout(IN := FALSE);

                tonSheetStackDischarge(
                    IN := TRUE,
                    PT := machineConfig.sheetStackDischargeTime
                );

                IF tonSheetStackDischarge.Q THEN

                    tonSheetStackDischarge(IN := FALSE);

                    sheetStackDischargeConveyorRunRequest := FALSE;

                    sheetStackDischargeControlState := 40;

                END_IF

            END_IF


        40: // START_RETURN_POSITIONING
            sheetStackDischargeState := 'START_RETURN';
            sheetStackDischargeStateCode := 40;

            sheetStackDischargeActive := TRUE;

            sheetStackDischargeConveyorRunRequest := FALSE;

            tonSheetStackDischarge(IN := FALSE);
            tonSheetStackDischargeStepTimeout(IN := FALSE);

            // EN: Request backstop return to the latched programmed target.
            //     The override remains active until the backstop returns.
            backstopTargetOverrideActive := TRUE;
            backstopTargetOverridePositionMm :=
                backstopProgrammedDischargeTargetMm;

            // EN: Request conveyor leveler to return down.
            //     The sequence does not wait for leveler feedback.
            conveyorLevelerTargetOverrideActive := TRUE;
            conveyorLevelerTargetOverridePositionMm :=
                machineConfig.conveyorLevelerMinPositionMm;

            sheetStackDischargeControlState := 50;


        50: // WAIT_BACKSTOP_RETURN
            sheetStackDischargeState := 'WAIT_BACKSTOP_RETURN';
            sheetStackDischargeStateCode := 50;

            sheetStackDischargeActive := TRUE;

            sheetStackDischargeConveyorRunRequest := FALSE;

            // EN: Keep backstop return target active.
            backstopTargetOverrideActive := TRUE;
            backstopTargetOverridePositionMm :=
                backstopProgrammedDischargeTargetMm;

            // EN: Keep conveyor leveler return target active.
            //     Feedback is intentionally ignored for sequence progress.
            conveyorLevelerTargetOverrideActive := TRUE;
            conveyorLevelerTargetOverridePositionMm :=
                machineConfig.conveyorLevelerMinPositionMm;

            // EN: If backstop is not in auto, do not wait for it.
            IF NOT backstopAutoCmd THEN

                sheetStackDischargeCycleHasManualSkip := TRUE;

                tonSheetStackDischargeStepTimeout(IN := FALSE);

                sheetStackDischargeControlState := 60;


            ELSIF backstopInPosition THEN

                tonSheetStackDischargeStepTimeout(IN := FALSE);

                sheetStackDischargeControlState := 60;


            ELSE

                tonSheetStackDischargeStepTimeout(
                    IN := TRUE,
                    PT := machineConfig.sheetStackDischargeReturnTimeout
                );

                IF tonSheetStackDischargeStepTimeout.Q THEN

                    // EN: Do not stay trapped waiting for return.
                    tonSheetStackDischargeStepTimeout(IN := FALSE);

                    sheetStackDischargeCycleHasTimeout := TRUE;

                    sheetStackDischargeFault := TRUE;
                    sheetStackDischargeFaultCode := 50;

                    sheetStackDischargeLastCycleOk := FALSE;
                    sheetStackDischargeLastResultCode := 3;
                    sheetStackDischargeLastFaultStepCode := 50;
                    sheetStackDischargeLastFaultCode := 50;

                    sheetStackDischargeControlState := 60;

                END_IF

            END_IF


        60: // FINISH
            sheetStackDischargeState := 'FINISH';
            sheetStackDischargeStateCode := 60;

            sheetStackDischargeActive := FALSE;
            sheetStackDischargePending := FALSE;
            sheetStackDischargeFinished := TRUE;

            sheetStackDischargeConveyorRunRequest := FALSE;

            backstopTargetOverrideActive := FALSE;
            conveyorLevelerTargetOverrideActive := FALSE;

            tonSheetStackDischarge(IN := FALSE);
            tonSheetStackDischargeStepTimeout(IN := FALSE);

            IF sheetStackDischargeCycleHasTimeout THEN

                sheetStackDischargeLastCycleOk := FALSE;
                sheetStackDischargeLastResultCode := 3;

                // EN: Keep manual intervention memory after timeout.
                //     The backstop may not have returned correctly.

            ELSIF sheetStackDischargeCycleHasManualSkip THEN

                sheetStackDischargeLastCycleOk := FALSE;
                sheetStackDischargeLastResultCode := 2;
                sheetStackDischargeLastFaultStepCode := 0;
                sheetStackDischargeLastFaultCode := 0;

                sheetStackDischargeFault := FALSE;
                sheetStackDischargeFaultCode := 0;

                // EN: Keep manual intervention memory because the backstop
                //     was not controlled automatically.


            ELSE

                sheetStackDischargeLastCycleOk := TRUE;
                sheetStackDischargeLastResultCode := 1;
                sheetStackDischargeLastFaultStepCode := 0;
                sheetStackDischargeLastFaultCode := 0;

                sheetStackDischargeFault := FALSE;
                sheetStackDischargeFaultCode := 0;

                // EN: Cycle completed correctly and backstop returned to
                //     programmed target. Clear manual intervention memory.
                backstopManualInterventionActive := FALSE;
                backstopManualInterventionPositionMm := 0.0;

            END_IF

            // EN: Always return to IDLE automatically.
            sheetStackDischargeControlState := 0;


    ELSE

        sheetStackDischargeControlState := 0;

    END_CASE;

END_IF;
END_METHOD

//==============================================================
// SIMPLE STACKER — SHEET STACK DISCHARGE CONVEYOR CONTROL
// EN: Controls the sheet stack discharge conveyor.
//     Conveyor runs while manual button is pressed or while
//     automatic request is active and conveyor automatic mode is enabled.
//
// Fault code
// 0 = No fault
// 1 = Safety circuit not OK
// 2 = Discharge conveyor drive not OK
//==============================================================
METHOD _SheetStackDischargeConveyorControl
VAR
    manualRunRequest   : BOOL;
    automaticRunRequest: BOOL;
    finalRunRequest    : BOOL;
END_VAR
//==============================================================
// SIMPLE STACKER — SHEET STACK DISCHARGE CONVEYOR CONTROL
// EN: Controls the sheet stack discharge conveyor in manual pulse
//     or automatic sequence request.
//==============================================================


//==============================================================
// 1) Default outputs
//==============================================================
sheetStackDischargeConveyorRun := FALSE;
sheetStackDischargeConveyorSpeedRefMPM := 0.0;


//==============================================================
// 2) Run request selection
//==============================================================
// EN: Manual command is momentary. Conveyor runs while button is pressed.
manualRunRequest :=
    sheetStackDischargeConveyorManualRunCmd;


// EN: Automatic request is generated by the discharge sequence.
//     This conveyor is assumed to be available for automatic cycle
//     whenever the master system is enabled.
automaticRunRequest :=
    sheetStackDischargeConveyorRunRequest;


// EN: Master system enable blocks both manual and automatic movement.
finalRunRequest :=
    systemRunEnable AND
    (
        manualRunRequest OR
        automaticRunRequest OR
		backstopHomeRunning
    );


//==============================================================
// 3) Fault detection
//==============================================================
IF NOT safetyCircuitOk THEN

    sheetStackDischargeConveyorState := 'SAFETY_OFF';

    sheetStackDischargeConveyorFault := TRUE;
    sheetStackDischargeConveyorFaultCode := 1;


ELSIF NOT sheetStackDischargeConveyorDriveOk THEN

    sheetStackDischargeConveyorState := 'DRIVE_NOT_OK';

    sheetStackDischargeConveyorFault := TRUE;
    sheetStackDischargeConveyorFaultCode := 2;


ELSE

    //==============================================================
    // 4) Fault reset
    //==============================================================
    IF resetCmd THEN

        sheetStackDischargeConveyorFault := FALSE;
        sheetStackDischargeConveyorFaultCode := 0;

    END_IF;


    //==============================================================
    // 5) Conveyor output control
    //==============================================================
    IF sheetStackDischargeConveyorFault THEN

        sheetStackDischargeConveyorState := 'FAULT';

        sheetStackDischargeConveyorRun := FALSE;
        sheetStackDischargeConveyorSpeedRefMPM := 0.0;


    ELSIF NOT systemRunEnable THEN

        // EN: Master stop disables movement without generating a conveyor fault.
        sheetStackDischargeConveyorState := 'SYSTEM_DISABLED';

        sheetStackDischargeConveyorRun := FALSE;
        sheetStackDischargeConveyorSpeedRefMPM := 0.0;


    ELSIF finalRunRequest THEN

        IF automaticRunRequest THEN

            sheetStackDischargeConveyorState := 'AUTO_RUN';

        ELSE

            sheetStackDischargeConveyorState := 'MANUAL_RUN';

        END_IF;

        sheetStackDischargeConveyorRun := TRUE;

        sheetStackDischargeConveyorSpeedRefMPM :=
            LIMIT(
                0.0,
                machineConfig.sheetStackDischargeConveyorSpeedMPM,
                machineConfig.maximumSpeedMPM
            );


    ELSE

        sheetStackDischargeConveyorState := 'STOP';

        sheetStackDischargeConveyorRun := FALSE;
        sheetStackDischargeConveyorSpeedRefMPM := 0.0;

    END_IF

END_IF;
END_METHOD

//==============================================================
// SIMPLE STACKER — SYSTEM CONTROL
// EN: Master system run enable and automatic homing requests.
//==============================================================
METHOD _SystemControl

//==============================================================
// 1) Edge detection
//==============================================================
rStartCmd := startCmd AND NOT startCmdOld;
startCmdOld := startCmd;

rStopCmd := stopCmd AND NOT stopCmdOld;
stopCmdOld := stopCmd;



//==============================================================
// 2) Stop machine pulse on critical fault
//==============================================================
stopMachineFaultCondition :=
    NOT safetyCircuitOk OR
    NOT sheetConveyor1DriveOk OR
    NOT sheetConveyor2DriveOk OR
    NOT sheetConveyor3DriveOk OR
    NOT backstopDriveOk OR
    NOT conveyorLevelerDriveOk OR
    NOT sheetStackDischargeConveyorDriveOk;

rStopMachineFaultCondition :=
    stopMachineFaultCondition AND
    NOT stopMachineFaultConditionOld;

stopMachineFaultConditionOld :=
    stopMachineFaultCondition;

tpStopMachinePulse(
    IN := rStopMachineFaultCondition,
    PT := T#500MS
);

stopMachinePulse :=
    tpStopMachinePulse.Q;


//==============================================================
// 2) Default one-scan requests
//==============================================================
backstopAutoHomeRequest := FALSE;
conveyorLevelerAutoHomeRequest := FALSE;


//==============================================================
// 3) Master system run enable
//==============================================================
IF NOT safetyCircuitOk THEN

    systemRunEnable := FALSE;

ELSIF rStopCmd THEN

    systemRunEnable := FALSE;

ELSIF rStartCmd THEN

    systemRunEnable := TRUE;

END_IF;


//==============================================================
// 4) Automatic homing on system start
//==============================================================
// EN: Auto-home is generated only on the rising edge of startCmd.
//     Each axis must be enabled in automatic mode.
//     This prevents automatic movement of axes intentionally left in manual.
IF rStartCmd AND systemRunEnable THEN

    // Backstop auto-home
    IF backstopAutoCmd AND
       NOT backstopHomed AND
       NOT backstopFault THEN

        backstopAutoHomeRequest := TRUE;

    END_IF;


    // Conveyor leveler auto-home
    IF conveyorLevelerAutoCmd AND
       NOT conveyorLevelerHomed AND
       NOT conveyorLevelerFault THEN

        conveyorLevelerAutoHomeRequest := TRUE;

    END_IF;

END_IF;
END_METHOD

END_FUNCTION_BLOCK

// ---- Library/Machine/Stacker/Cpx/FB_ComplexSheetStackerControl.TcPOU
FUNCTION_BLOCK FB_ComplexSheetStackerControl
VAR_INPUT

    //==============================================================
    // Group command inputs
    //==============================================================
    startCmd                            : BOOL;
    stopCmd                             : BOOL;
    resetCmd                            : BOOL;


    //==============================================================
    // Speed reference inputs
    //==============================================================
    lineSpeedMPM                        : REAL;

    // EN: Current sheet length [mm].
    // PT: Comprimento atual da chapa [mm].
    sheetLengthMm                       : REAL;


    //==============================================================
    // Package command input
    //==============================================================
    // EN: Maintained automatic unload request from the production metrics.
    //     It is accepted only once and is rearmed after the command turns FALSE.
    // PT: Pedido automático mantido de descarga vindo das métricas de produção.
    //     É aceito apenas uma vez e rearmado após o comando ficar FALSE.
    packageCompleteCmd                  : BOOL;

    // EN: Rising edge requests a complete discharge cycle for batch change.
    // PT: Borda de subida solicita um ciclo completo de descarte para troca de lote.
    changeBatchCmd                      : BOOL;

	// EN: Local unload request accepted on the rising edge.
	// PT: Pedido local de descarga aceito na borda de subida.
	stackerUnloadCmd                     : BOOL;

	sheetConveyorsSpeedUpCmd : BOOL;

    //==============================================================
    // Machine configuration
    //==============================================================
    machineConfig                       : ComplexStackerConfig_TypeStruct;


    //==============================================================
    // Safety input
    //==============================================================
    safetyCircuitOk                     : BOOL;


    //==============================================================
    // Synchronized conveyor drive status inputs
    //==============================================================
    sheetConveyor1DriveOk               : BOOL;
    sheetConveyor2DriveOk               : BOOL;
    sheetConveyor3DriveOk               : BOOL;
    sheetConveyor4DriveOk               : BOOL;
    elevatorDriveOk              : BOOL;


    //==============================================================
    // Auxiliary drive status inputs
    //==============================================================
    backstopDriveOk                     : BOOL;

	//==============================================================
	// Sheet stack discharge conveyor drive status input
	//==============================================================
    sheetStackDischargeConveyorDriveOk                 : BOOL;

	//==============================================================
	// EN: Stack buffer conveyor drive status inputs
	// PT: Entradas de estado dos acionamentos das esteiras buffer
	//==============================================================
	stackBufferConveyor1DriveOk            : BOOL;
	stackBufferConveyor2DriveOk            : BOOL;
	stackBufferConveyor3DriveOk            : BOOL;

	//==============================================================
	// EN: Stack detection sensors
	// PT: Sensores de detecção das pilhas
	//==============================================================
	stackBufferConveyor1StackPresentSensor : BOOL;
	stackBufferConveyor2StackPresentSensor : BOOL;
	stackBufferConveyor3StackPresentSensor : BOOL;
	elevatorStackPresentSensor             : BOOL;
	elevatorStackExitClearSensor           : BOOL;
	backstopMaterialInterlockSensor         : BOOL;
	backstopStackLevelSensor                : BOOL;

	
    //==============================================================
    // Position / measurement inputs
    //==============================================================
    stackHeightMm                       : REAL;
    backstopPositionMm                  : REAL;
    elevatorPositionMm           : REAL;


	//==============================================================
	// Elevator command inputs
	//==============================================================
	// EN: Starts elevator homing cycle.
	// PT: Inicia o ciclo de homing do elevador.
	elevatorHomeCmd              : BOOL;
	
	// EN: Enables elevator automatic mode. Auto-home is requested on
	//     startCmd and automatic leveling uses the stack level sensor.
	// PT: Habilita o modo automático do elevador. O auto-home é solicitado
	//     no startCmd e o nivelamento automático usa o sensor de nível da pilha.
	elevatorAutoCmd              : BOOL;
	
	// EN: Jog-up command in manual mode or during automatic leveling.
	// PT: Comando de jog para subir no manual ou durante o nivelamento automático.
	elevatorUpCmd                : BOOL;
	
	// EN: Jog-down command in manual mode or during automatic leveling.
	// PT: Comando de jog para descer no manual ou durante o nivelamento automático.
	elevatorDownCmd              : BOOL;


    //==============================================================
    // Elevator limit inputs
    //==============================================================
    elevatorUpperSafetyLimit     : BOOL;
    elevatorLowerSafetyLimit     : BOOL;

    elevatorUpperLimit           : BOOL;
    elevatorLowerLimit           : BOOL;


    //==============================================================
    // Backstop command inputs
    //==============================================================
    // EN: Starts the backstop homing cycle.
    // PT: Inicia o ciclo de homing do backstop.
    backstopHomeCmd                     : BOOL;
	
    // EN: Starts the backstop homing cycle.
    // PT: Inicia o ciclo de homing do backstop.
    backstopExecutePositioningCmd			 : BOOL;
    // EN: Enables automatic positioning according to sheet length.
    // PT: Habilita posicionamento automático conforme comprimento da chapa.
    backstopAutoCmd                     : BOOL;

    // EN: Manual open command.
    // PT: Comando manual para abrir.
    backstopOpenCmd                     : BOOL;

    // EN: Manual close command.
    // PT: Comando manual para fechar.
    backstopCloseCmd                    : BOOL;


    //==============================================================
    // Backstop limit inputs
    //==============================================================
    backstopSafeMaxLimit                    : BOOL;	
    backstopMaxLimit                 	   	: BOOL;
    backstopMinLimit                   		: BOOL;
    backstopSafeMinLimit                    : BOOL;


    //==============================================================
    // Sheet handling command inputs
    //==============================================================
	sheetStackDischargeConveyorManualRunCmd : BOOL;
    noCrushRollersDownCmd                 	: BOOL;

	// EN: Runs all three stack buffer conveyors.
	// PT: Aciona as três esteiras buffer de pilhas.
	stackBufferConveyorsRunCmd               : BOOL;

	// EN: Enables automatic operation of the sheet stack alignment brush.
	// PT: Habilita a operação automática da escova de alinhamento da pilha.
	sheetStackAlignmentBrushEnableCmd        : BOOL;

	//==============================================================
	// Input / Entrada
	//==============================================================
	paperPressAutoManCmd : BOOL;

	// EN: Enables automatic operation of the exhaust fan installed
	//     on sheet conveyor 1.
	// PT: Habilita a operação automática do exaustor instalado
	//     na esteira de chapas 1.
	sheetConveyor1ExhaustFanCmd : BOOL;

	//==============================================================
	// EN: Independent sheet brush commands
	// PT: Comandos independentes das escovas de chapas
	//==============================================================
	sheetBrush1Cmd       : BOOL;
	sheetBrush2Cmd       : BOOL;
	sheetBrush3Cmd       : BOOL;
	sheetBrush4Cmd       : BOOL;
	sheetBrushAutoManCmd : BOOL;
	
	safetyFeedBack1 	: BOOL;
	safetyFeedBack2 	: BOOL;
	safetyFeedBack3 	: BOOL;
	safetyFeedBack4 	: BOOL;
	safetyFeedBack5 	: BOOL;
	safetyFeedBack6 	: BOOL;
	safetyFeedBack7 	: BOOL;
	safetyFeedBack8 	: BOOL;	
	safetyFeedBack9 	: BOOL;	
	safetyFeedBack10 	: BOOL;		
			

END_VAR


VAR_OUTPUT

	hmiAlarms : hmiAlarmsComplexStacker_TypeStruct;
	hmiStatus : hmiStatusComplexStacker_TypeStruct;
	stackerRunning : BOOL;
	alarmActive	: BOOL;
	stopMachinePulse : BOOL;
	reset 	: BOOL;

	// EN: TRUE during an accepted unload sequence or while a stacker axis
	//     executes homing. Intended to command an external warning siren.
	// PT: TRUE durante uma sequência de descarga aceita ou enquanto um eixo
	//     do stacker executa homing. Destinada ao comando de uma sirene externa.
	stackerBuzzer1 : BOOL;
	stackerBuzzer2 : BOOL;
	// EN: One-scan pulse generated when a local unload request is accepted.
	//     It can be used to reset the external pile quantity in Metrics.
	// PT: Pulso de um ciclo gerado quando um pedido local de descarga é aceito.
	//     Pode ser usado para resetar a quantidade externa da pilha no Metrics.
	stackerUnloadAccepted : BOOL;

	// EN: 20 ms pulse used to reset the external stack counter.
	// PT: Pulso de 20 ms usado para resetar o contador externo de pilhas.
	externalCounterReset : BOOL;

    //==============================================================
    // Synchronized conveyor drive outputs
    //==============================================================
    sheetConveyor1Run                   : BOOL;
    sheetConveyor2Run                   : BOOL;
    sheetConveyor3Run                   : BOOL;
    sheetConveyor4Run                   : BOOL;

	// EN: Sheet conveyor 1 exhaust fan run command.
	// PT: Comando de acionamento do exaustor da esteira de chapas 1.
	sheetConveyor1ExhaustFanRun           : BOOL;
	
	//==============================================================
	// Elevator drive outputs
	//==============================================================
	// EN: Elevator up run command.
	// PT: Comando para subir o elevador.
	elevatorRunUp                : BOOL;
	
	// EN: Elevator down run command.
	// PT: Comando para descer o elevador.
	elevatorRunDown              : BOOL;
	
	//==============================================================
	// Elevator magnetic brake output
	//==============================================================
	// EN: Magnetic brake release output. TRUE = brake released.
	// PT: Saída de liberação do freio magnético. TRUE = freio liberado.
	elevatorBrakeRelease         : BOOL;	

	// EN: Enables the elevator servo together with the stacker control.
	//     The servo remains enabled while stopped with zero speed reference.
	// PT: Habilita o servo do elevador junto com o controle do stacker.
	//     O servo permanece habilitado quando parado com referência zero.
	elevatorDriveEnable          : BOOL;

    //==============================================================
    // Backstop drive outputs
    //==============================================================
    // EN: Backstop forward run command. Positive/opening direction.
    // PT: Comando frente do backstop. Direção positiva/abrir.
    backstopRunFw                       : BOOL;

    // EN: Backstop reverse run command. Negative/closing direction.
    // PT: Comando reverso do backstop. Direção negativa/fechar.
    backstopRunRev                      : BOOL;

    // EN: Enables the backstop servo together with the stacker control.
    // PT: Habilita o servo do backstop junto com o controle do stacker.
    backstopDriveEnable                 : BOOL;

	//==============================================================
	// Sheet stack discharge conveyor outputs
	//==============================================================
	// EN: Sheet stack discharge conveyor run command.
	// PT: Comando de giro da esteira de descarga da pilha.
	sheetStackDischargeConveyorRun          : BOOL;

	//==============================================================
	// EN: Stack buffer conveyor run outputs
	// PT: Saídas de acionamento das esteiras buffer de pilhas
	//==============================================================
	stackBufferConveyor1Run                 : BOOL;
	stackBufferConveyor2Run                 : BOOL;
	stackBufferConveyor3Run                 : BOOL;




    //==============================================================
    // Synchronized conveyor speed reference outputs
    //==============================================================
    sheetConveyor1SpeedRefMPM           : REAL;
    sheetConveyor2SpeedRefMPM           : REAL;
    sheetConveyor3SpeedRefMPM           : REAL;
    sheetConveyor4SpeedRefMPM           : REAL;

    // EN: Signed elevator speed reference [mm/s]. Positive moves up
    //     and negative moves down.
    // PT: Referência de velocidade com sinal do elevador [mm/s].
    //     Positivo sobe e negativo desce.
    elevatorSpeedRefMmps                 : REAL;
	// EN: Sheet stack discharge conveyor speed reference [m/min].
	// PT: Referência de velocidade da esteira de descarga da pilha [m/min].
	sheetStackDischargeConveyorSpeedRefMPM  : REAL;

	// EN: Stack buffer conveyor speed references [m/min].
	// PT: Referências de velocidade das esteiras buffer [m/min].
	stackBufferConveyor1SpeedRefMPM         : REAL;
	stackBufferConveyor2SpeedRefMPM         : REAL;
	stackBufferConveyor3SpeedRefMPM         : REAL;

	// EN: TRUE while all three stack buffer positions are occupied.
	// PT: TRUE enquanto as três posições buffer estiverem ocupadas.
	stackBufferFull                         : BOOL;

	// EN: Requests the parent controller to reduce the machine speed.
	// PT: Solicita ao controlador pai a redução da velocidade da máquina.
	lineSpeedReductionRequest               : BOOL;

    //==============================================================
    // Backstop speed reference output
    //==============================================================
    // EN: Signed backstop speed reference [mm/s]. Positive opens and negative closes.
    // PT: Referência de velocidade com sinal do backstop [mm/s]. Positivo abre e negativo fecha.
    backstopSpeedRefMmps                : REAL;
	
	
	
    backstopPlateUpSolenoid                : BOOL;


    //==============================================================
    // Backstop encoder set outputs
    //==============================================================
    // EN: Pulse output to set/reset backstop encoder position.
    // PT: Pulso de saída para setar/resetar a posição do encoder do backstop.
    backstopSetEncoderPosition          : BOOL;

    // EN: Position value to set in the encoder block [mm].
    // PT: Valor de posição a ser gravado no bloco do encoder [mm].
    backstopSetEncoderPositionMm        : REAL;


    //==============================================================
    // Pneumatic valve outputs
    //==============================================================
    brakeValve                          : BOOL;

    sheetBrush1Valve                    : BOOL;
    sheetBrush2Valve                    : BOOL;
    sheetBrush3Valve                    : BOOL;
    sheetBrush4Valve                    : BOOL;

    brakeBrushValve                     : BOOL;
    backstopUpValve                     : BOOL;
    noCrushRollersUpDownValve               : BOOL;

	// EN: Sheet stack alignment brush command. TRUE = lowered/engaged;
	//     FALSE = raised/disengaged.
	// PT: Comando da escova de alinhamento da pilha. TRUE = abaixada/acionada;
	//     FALSE = levantada/desacionada.
	sheetStackAlignmentBrush              : BOOL;

	paperPressSolenoid : BOOL;
    //==============================================================
    // General status outputs
    //==============================================================
    deviceState                         : STRING(30);

    faultActive                         : BOOL;
    synchronizedConveyorsRunning        : BOOL;


    //==============================================================
    // Sheet stack separation status outputs
    //==============================================================
    sheetStackSeparationState           : STRING(30);
    sheetStackSeparationStateCode       : INT;

    sheetStackSeparationReady           : BOOL;
    sheetStackSeparationActive          : BOOL;

    // EN: One-scan pulse when sheet stack separation starts.
    // PT: Pulso de um ciclo quando inicia a separação da pilha de chapas.
    sheetStackSeparationStarted         : BOOL;

    // EN: One-scan pulse when sheet stack separation finishes.
    // PT: Pulso de um ciclo quando finaliza a separação da pilha de chapas.
    sheetStackSeparationFinished        : BOOL;

    // EN: Brake active during sheet stack separation.
    // PT: Freio ativo durante a separação da pilha de chapas.
    sheetStackBrakeActive               : BOOL;


    //==============================================================
    // Sheet conveyor 2 separation status outputs
    //==============================================================
    sheetConveyor2SeparationActive      : BOOL;

    // EN: One-scan pulse when conveyor 2 separation tracking starts.
    // PT: Pulso de um ciclo quando inicia o rastreamento de separação da esteira 2.
    sheetConveyor2SeparationStarted     : BOOL;

    // EN: One-scan pulse when conveyor 2 separation tracking finishes.
    // PT: Pulso de um ciclo quando finaliza o rastreamento de separação da esteira 2.
    sheetConveyor2SeparationFinished    : BOOL;

    sheetConveyor2HighSpeedActive       : BOOL;

    // EN: Current conveyor 2 separation tracking distance [m].
    // PT: Distância atual rastreada na separação da esteira 2 [m].
    sheetConveyor2TrackingDistanceM     : REAL;

    // EN: Conveyor 2 separation target distance [m].
    // PT: Distância alvo de separação da esteira 2 [m].
    sheetConveyor2TargetDistanceM       : REAL;


    //==============================================================
    // Sheet conveyor 3 separation status outputs
    //==============================================================
    sheetConveyor3SeparationActive      : BOOL;

    // EN: One-scan pulse when conveyor 3 separation tracking starts.
    // PT: Pulso de um ciclo quando inicia o rastreamento de separação da esteira 3.
    sheetConveyor3SeparationStarted     : BOOL;

    // EN: One-scan pulse when conveyor 3 separation tracking finishes.
    // PT: Pulso de um ciclo quando finaliza o rastreamento de separação da esteira 3.
    sheetConveyor3SeparationFinished    : BOOL;

    sheetConveyor3HighSpeedActive       : BOOL;

    // EN: Current conveyor 3 separation tracking distance [m].
    // PT: Distância atual rastreada na separação da esteira 3 [m].
    sheetConveyor3TrackingDistanceM     : REAL;

    // EN: Conveyor 3 separation target distance [m].
    // PT: Distância alvo de separação da esteira 3 [m].
    sheetConveyor3TargetDistanceM       : REAL;

    //==============================================================
    // Sheet conveyor 4 separation status outputs
    //==============================================================
    sheetConveyor4SeparationActive      : BOOL;
    sheetConveyor4SeparationStarted     : BOOL;
    sheetConveyor4SeparationFinished    : BOOL;
    sheetConveyor4HighSpeedActive       : BOOL;
    sheetConveyor4TrackingDistanceM     : REAL;
    sheetConveyor4TargetDistanceM       : REAL;

	//==============================================================
	// Elevator encoder set outputs
	//==============================================================
	// EN: Pulse output to set/reset elevator encoder position.
	// PT: Pulso de saída para setar/resetar a posição do encoder do elevador.
	elevatorSetEncoderPosition   : BOOL;
	
	// EN: Position value to set in the elevator encoder block [mm].
	// PT: Valor de posição a ser gravado no bloco do encoder do elevador [mm].
	elevatorSetEncoderPositionMm : REAL;
	
	
	//==============================================================
	// Elevator status outputs
	//==============================================================
	elevatorState                : STRING(30);
	
	elevatorHomed                : BOOL;
	elevatorInPosition           : BOOL;

	// EN: TRUE when the homed elevator is at or below the configured
	//     minimum position considering the position tolerance.
	// PT: TRUE quando o elevador referenciado está na posição mínima
	//     configurada ou abaixo dela, considerando a tolerância.
	elevatorAtMinPosition        : BOOL;

	// EN: TRUE when the homed elevator is at or above the configured
	//     maximum position considering the position tolerance.
	// PT: TRUE quando o elevador referenciado está na posição máxima
	//     configurada ou acima dela, considerando a tolerância.
	elevatorAtMaxPosition        : BOOL;

	// EN: TRUE while manual jog speed is reduced near the endpoint
	//     toward which the elevator is moving.
	// PT: TRUE enquanto a velocidade do jog manual estiver reduzida próximo
	//     da extremidade para a qual o elevador está se movimentando.
	elevatorManualLowSpeedZoneActive : BOOL;

	elevatorFault                : BOOL;
	elevatorFaultCode            : INT;
	
	// EN: Current calculated elevator target position [mm].
	// PT: Posição alvo calculada atual do elevador [mm].
	elevatorTargetPositionMm     : REAL;
	
	// EN: Current elevator position error [mm].
	// PT: Erro atual de posição do elevador [mm].
	elevatorPositionErrorMm      : REAL;

    //==============================================================
    // Backstop status outputs
    //==============================================================
    backstopState                       : STRING(30);

    backstopHomed                       : BOOL;
    backstopInPosition                  : BOOL;
    backstopFault                       : BOOL;
    backstopFaultCode                   : INT;

    // EN: Current calculated target position [mm].
    // PT: Posição alvo calculada atualmente [mm].
    backstopTargetPositionMm            : REAL;

    // EN: Current position error [mm].
    // PT: Erro atual de posição [mm].
    backstopPositionErrorMm             : REAL;
	
	//==============================================================
	// Sheet stack discharge conveyor control state
	//==============================================================
	sheetStackDischargeConveyorState               : STRING(30);
	sheetStackDischargeConveyorFault               : BOOL;
	sheetStackDischargeConveyorFaultCode           : INT;
	
	//==============================================================
	// Sheet stack discharge sequence status outputs
	//==============================================================
	sheetStackDischargeState                : STRING(30);
	sheetStackDischargeStateCode            : INT;
	
	sheetStackDischargePending              : BOOL;
	sheetStackDischargeActive               : BOOL;
	sheetStackDischargeStarted              : BOOL;
	sheetStackDischargeFinished             : BOOL;
	
	sheetStackDischargeFault                : BOOL;
	sheetStackDischargeFaultCode            : INT;
	
	//==============================================================
	// Sheet stack discharge last cycle diagnostic outputs
	//==============================================================
	sheetStackDischargeLastCycleOk          : BOOL;
	sheetStackDischargeLastResultCode       : INT;
	sheetStackDischargeLastFaultStepCode    : INT;
	sheetStackDischargeLastFaultCode        : INT;	

	// EN: Requests a CiA 402 quick stop while the servo disable delay is active.
	// PT: Solicita o quick stop CiA 402 durante o atraso de desabilitação do servo.
	elevatorQuickStop                       : BOOL;

END_VAR

VAR
	
	//==============================================================
	// Stop machine pulse control
	//==============================================================
	stopMachineFaultCondition     : BOOL;
	stopMachineFaultConditionOld  : BOOL;
	rStopMachineFaultCondition    : BOOL;
	
	tpStopMachinePulse            : TP;
	
	//==============================================================
	// Backstop manual intervention memory
	//==============================================================
	backstopManualInterventionActive     : BOOL;
	backstopManualInterventionPositionMm : REAL;
	
	//==============================================================
	// Sheet stack discharge backstop latched targets
	//==============================================================
	backstopProgrammedDischargeTargetMm : REAL;
	backstopDischargeOpenBasePositionMm : REAL;
	backstopDischargeOpenTargetMm       : REAL;
	
	//==============================================================
	// Backstop automatic positioning command control
	//==============================================================
	backstopExecutePositioningCmdOld    : BOOL;
	rBackstopExecutePositioning         : BOOL;
	
	backstopTargetOverrideOld           : BOOL;
	backstopTargetOverrideFallingEdge   : BOOL;
	
	backstopPositioningRequestActive    : BOOL;
	backstopLatchedTargetPositionMm     : REAL;
	backstopProgrammedTargetPositionMm  : REAL;
	
	//==============================================================
	// Backstop manual intervention memory
	//==============================================================
	// EN: Used by automatic discharge sequence to avoid closing onto material
	//     after operator manual intervention.

	//==============================================================
	// Backstop encoder set pulse
	//==============================================================
	backstopSetEncoderPositionTrigger  : BOOL;
	tpBackstopSetEncoderPosition       : TP;

	//==============================================================
	// Sheet stack discharge backstop latched targets
	//==============================================================

    //==============================================================
    // Group state machine
    //==============================================================
    syncConveyorsState                  : INT;


    //==============================================================
    // Package separation state machine
    //==============================================================
    packageSeparationState              : INT;


    //==============================================================
    // Backstop state machine
    //==============================================================
    backstopControlState                : INT;


    //==============================================================
    // Edge detection
    //==============================================================
    startCmdOld                         : BOOL;
    stopCmdOld                          : BOOL;

	// EN: Locks the maintained automatic request after it is accepted.
	// PT: Bloqueia o pedido automático mantido após ele ser aceito.
	packageCompleteCmdAcceptedLatch       : BOOL;
	changeBatchCmdOld                     : BOOL;
	changeBatchRequestPending             : BOOL;
	changeBatchCycleActive                : BOOL;

	// EN: Local unload command rising-edge detection.
	// PT: Detecção de borda de subida do comando local de descarga.
	stackerUnloadCmdOld                   : BOOL;
	rStackerUnloadCmd                     : BOOL;

	// EN: Internal one-scan event generated for any accepted unload source.
	// PT: Evento interno de um scan gerado para qualquer fonte de descarga aceita.
	dischargeRequestAccepted              : BOOL;

    backstopHomeCmdOld                  : BOOL;


    //==============================================================
    // Internal conditions
    //==============================================================
    allSynchronizedDrivesOk             : BOOL;
    anyFault                            : BOOL;
    speedControlEnabled                 : BOOL;
    rampReset                           : BOOL;


    //==============================================================
    // Sheet length conversion
    //==============================================================
    // EN: Internal sheet length converted from mm to m.
    // PT: Comprimento interno da chapa convertido de mm para m.
    sheetLengthM                        : REAL;


    //==============================================================
    // Normal speed calculation
    //==============================================================
    effectiveLineSpeedMPM                : REAL;
    normalStackerSpeedMPM               : REAL;

    sheetConveyor1NormalSpeedMPM        : REAL;
    sheetConveyor2NormalSpeedMPM        : REAL;
    sheetConveyor3NormalSpeedMPM        : REAL;
    sheetConveyor4NormalSpeedMPM        : REAL;
    elevatorNormalSpeedMPM       : REAL;


    //==============================================================
    // Package gap speed calculation
    //==============================================================
    sheetConveyor1GapSpeedMPM           : REAL;
    sheetConveyor2GapSpeedMPM           : REAL;
    sheetConveyor3GapSpeedMPM           : REAL;
    sheetConveyor4GapSpeedMPM           : REAL;


    //==============================================================
    // Speed targets
    //==============================================================
    sheetConveyor1TargetSpeedMPM        : REAL;
    sheetConveyor2TargetSpeedMPM        : REAL;
    sheetConveyor3TargetSpeedMPM        : REAL;
    sheetConveyor4TargetSpeedMPM        : REAL;
    elevatorTargetSpeedMPM       : REAL;


    //==============================================================
    // Package gap distance calculation
    //==============================================================
    packageGapDistanceTargetM           : REAL;

    sheetConveyor2OpeningSpeedMPM       : REAL;
    sheetConveyor3OpeningSpeedMPM       : REAL;
    sheetConveyor4OpeningSpeedMPM       : REAL;

    sheetConveyor2OpeningDistanceM      : REAL;
    sheetConveyor3OpeningDistanceM      : REAL;
    sheetConveyor4OpeningDistanceM      : REAL;


	//==============================================================
	// Elevator state machine
	//==============================================================
	elevatorControlState         : INT;
	
	
	//==============================================================
	// Elevator edge detection
	//==============================================================
	elevatorHomeCmdOld           : BOOL;
	rElevatorHome                : BOOL;
	
	
	//==============================================================
	// Elevator encoder set pulse
	//==============================================================
	elevatorSetEncoderPositionTrigger   : BOOL;
	tpElevatorSetEncoderPosition        : TP;
	
	
	//==============================================================
	// Elevator control calculation
	//==============================================================
	elevatorAutoTargetPositionMm        : REAL;
	elevatorRawSpeedRefMmps             : REAL;
	
	// EN: Internal signed speed command. Positive = up, negative = down.
	// PT: Comando interno de velocidade com sinal. Positivo = subir, negativo = descer.
	elevatorSignedSpeedRefMmps          : REAL;
	
	elevatorAbsPositionErrorMm          : REAL;
	
	
	//==============================================================
	// Elevator movement permissions
	//==============================================================
	elevatorUpAllowed                   : BOOL;
	elevatorDownAllowed                 : BOOL;
	
	elevatorDriveEnableRequest          : BOOL;
	elevatorMoveRequest                 : BOOL;
	elevatorBrakeReleaseRequest         : BOOL;
	
	
	//==============================================================
	// Elevator homing
	//==============================================================
	elevatorHomeLimitReached            : BOOL;
	elevatorHomeDownAllowed             : BOOL;
	elevatorHomeReleaseAllowed          : BOOL;
	elevatorManualCommandArmed          : BOOL;
	elevatorManualCommandRequest        : BOOL;
	elevatorReadyForAutomaticCycle      : BOOL;

	// EN: Keeps the discharge conveyor active from the lower home limit until
	//     the minimum run time and platform-clear conditions are confirmed.
	// PT: Mantém a esteira de descarga ativa desde o limite inferior do home até
	//     confirmar o tempo mínimo de giro e as condições de plataforma livre.
	elevatorHomeDischargeConveyorRunRequest : BOOL;
	elevatorHomeDischargeComplete            : BOOL;
	
	
	//==============================================================
	// Elevator timers
	//==============================================================
	tonElevatorHomingTimeout            : TON;
	tonElevatorHomeSettleDelay          : TON;
	tonElevatorHomeDischargeMinimumRun  : TON;
	tonElevatorLevelingSpeed2Delay      : TON;

	// EN: Filters a brief backstop material interlock during an upward request.
	// PT: Filtra um acionamento breve do intertravamento de material durante a subida.
	tonElevatorUpBlockedByBackstopAlarm : TON;
	
	// EN: Delay after brake release before motor movement.
	// PT: Atraso após liberar o freio antes de movimentar o motor.
	tonElevatorBrakeReleaseDelay        : TON;
	
	// EN: Keeps brake released for a short time after movement stops.
	// PT: Mantém o freio liberado por um tempo após parar o movimento.
	tonElevatorBrakeHoldDelay           : TON;

	// EN: Keeps the servo enabled while the quick-stop command is processed.
	// PT: Mantém o servo habilitado durante o processamento do comando de quick stop.
	tofElevatorDriveDisableDelay        : TOF;
	
	
	//==============================================================
	// Elevator speed ramp instance
	//==============================================================
	// EN: Ramp used for elevator vertical speed [mm/s].
	// PT: Rampa usada para velocidade vertical do elevador [mm/s].
	instRampElevator                    : FB_Gen_SRamp;
	

    //==============================================================
    // Backstop control calculation
    //==============================================================
    backstopAutoTargetPositionMm        : REAL;
    backstopRawSpeedRefMmps             : REAL;
    backstopAbsPositionErrorMm          : REAL;

    backstopHomeLimitReached            : BOOL;
    backstopOpenAllowed                 : BOOL;
    backstopCloseAllowed                : BOOL;

    rBackstopHome                       : BOOL;


	//==============================================================
	// Backstop homing edge detection
	//==============================================================
	backstopHomeLimitOld                 : BOOL;
	backstopHomeLimitFallingEdge         : BOOL;
	backstopHomeMoveAllowed              : BOOL;
	
	
	
	//==============================================================
	// Backstop timers
	//==============================================================
	tonBackstopHomeSettleDelay           : TON;



    //==============================================================
    // Backstop timers
    //==============================================================
    tonBackstopHomingTimeout            : TON;


    //==============================================================
    // Speed ramp instances
    //==============================================================
    instRampSheetConveyor1              : FB_Gen_SRamp;
    instRampSheetConveyor2              : FB_Gen_SRamp;
    instRampSheetConveyor3              : FB_Gen_SRamp;
    instRampSheetConveyor4              : FB_Gen_SRamp;


    //==============================================================
    // PLC scan time measurement
    //==============================================================
    instCycleTime                       : CYCLE_TIME;
    scanTimeS                           : REAL;
    scanTimeMs                          : REAL;

	backstopSignedSpeedRefMmps: REAL;
	
	//==============================================================
	// Sheet stack discharge state machine
	//==============================================================
	sheetStackDischargeControlState         : INT;
	
	
	//==============================================================
	// Sheet stack discharge request pulse
	//==============================================================
	// EN: Extends an accepted unload event for the external counter reset.
	// PT: Prolonga um evento de descarga aceito para resetar o contador externo.
	tpExternalCounterReset                  : TP;
	
	
	//==============================================================
	// Sheet stack discharge timers
	//==============================================================
	tonSheetStackDischarge                  : TON;
	tonSheetStackDischargePlatformClearTimeout : TON;
	elevatorPlatformClearDetected           : BOOL;
	elevatorStackPresentAtDischargeStart    : BOOL;
	
	
	//==============================================================
	// Sheet stack discharge internal conditions
	//==============================================================
	sheetStackDischargeFaultCondition       : BOOL;

	// EN: Remembers that the alignment brush was raised for the current
	//     automatic discharge cycle.
	// PT: Memoriza que a escova de alinhamento foi levantada para o ciclo
	//     atual de descarga automática.
	sheetStackAlignmentBrushLiftedForDischarge : BOOL;
	
	
	//==============================================================
	// Backstop target override
	//==============================================================
	backstopTargetOverrideActive            : BOOL;
	backstopTargetOverridePositionMm        : REAL;
	backstopRequiredForAutomaticOperation   : BOOL;
	
	
	//==============================================================
	// Elevator target override
	//==============================================================
	elevatorTargetOverrideActive     : BOOL;
	elevatorTargetOverridePositionMm : REAL;	
	
	
	sheetStackDischargeConveyorRunRequest: BOOL;
	instTONBackstopDownDelay: TON;
	
	//==============================================================
	// Sheet stack discharge step timeout
	//==============================================================
	tonSheetStackDischargeStepTimeout       : TON;
	
	sheetStackDischargeCycleHasManualSkip   : BOOL;
	sheetStackDischargeCycleHasTimeout      : BOOL;	
	
	
	//==============================================================
	// Elevator homing edge detection
	//==============================================================
	elevatorHomeLimitOld                 : BOOL;
	elevatorHomeLimitFallingEdge         : BOOL;	

	//==============================================================
	// System master run control
	//==============================================================
	systemRunEnable : BOOL;
	
	rStartCmd : BOOL;
	rStopCmd  : BOOL;
	
	//==============================================================
	// Automatic homing requests generated by master start
	//==============================================================
	backstopAutoHomeRequest        : BOOL;
	elevatorAutoHomeRequest : BOOL;

	// EN: Latched start requests awaiting valid homing permissives.
	// PT: Pedidos de partida memorizados aguardando permissivos válidos de homing.
	backstopAutoHomePending        : BOOL;
	elevatorAutoHomePending        : BOOL;
	
	//==============================================================
	// Elevator home request command control
	//==============================================================
	elevatorHomeRequestCombined    : BOOL;
	elevatorHomeRequestCombinedOld : BOOL;
	backstopHomeRunning: BOOL;
	//==============================================================
	// Backstop home request command control
	//==============================================================
	backstopHomeRequestCombined    : BOOL;
	backstopHomeRequestCombinedOld : BOOL;

